# EPICS autosave request: tests/testfiles/cfg/SF_UPHS_PV.req
$(SYS):GAP_SP
$(SYS):PHI_SET
